TYPE UNION_DWORD_REAL :
UNION
    Value_Word 	: DWORD;
    Value_Real  : REAL;
END_UNION
END_TYPE

(* stored: Version 1.1.0.1, ProductVersion 3.1.4026.18
   DUT UNION_DWORD_REAL: Id {39cee267-2750-4bcd-8e56-1fd13e05b748} *)
